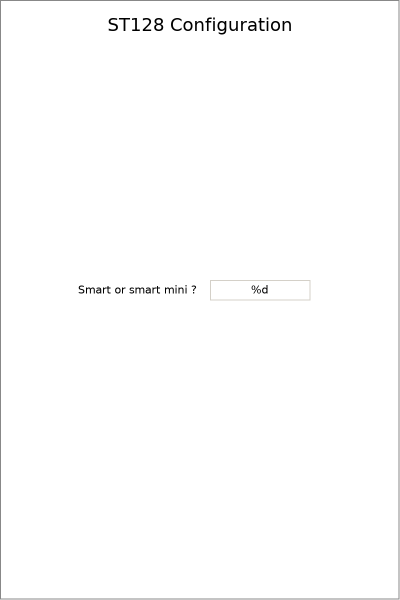
VISUALIZATION VISU_Recipe_ST128  // 400x600
    Label (0,5 400x40), "ST128 Configuration"
    Label (0,280 200x20), "Smart or smart mini ?"
    Textfield (210,280 100x20), "%d", text variable: _20_AUTO.recipe.st128.xIsTypeMiniOrSmart
        OnMouseDown: write the text variable via Default
END_VISUALIZATION

(* stored: Version 1.1.0.1, ProductVersion 3.1.4024.6
   Visu VISU_Recipe_ST128: Id {ae60a776-cc1a-4dd8-8512-5d3d6ebd2acf} *)
